PROGRAM LsBkgrdLsSerialCom
VAR_INPUT
	Config : LightspeedConfig;
END_VAR
VAR
END_VAR

// AttenuationFilterConfigs
IF Config.AttenuationFilterConfigs.FW212CAttenuationFilterConfig.IsEnabled OR 
   Config.AttenuationFilterConfigs.ELL14kAttenuationFilterConfig.IsEnabled OR
   Config.AttenuationFilterConfigs.ELL9AttenuationFilterConfig.IsEnabled THEN
	BkgrdSerialAttenuation();	
END_IF

// SliderAttenuationFilterConfigs
IF Config.SliderAttenuationFilterConfigs.ELL6SliderFilterConfig.IsEnabled THEN
	BkgrdSerialSliderAttenuation();	
END_IF

// RotatingSwitchConfigs
IF Config.RotatingSwitchConfigs.ELL18RotatingSwitchConfig.IsEnabled THEN
	BkgrdSerialRotatingSwitch();	
END_IF

// PolarisationFilterConfigs
IF Config.PolarisationFilterConfigs.FW212CPolarisationFilterConfig.IsEnabled OR 
   Config.PolarisationFilterConfigs.ELL14KPolarisationFilterConfig.IsEnabled THEN
	BkgrdSerialPolarisation();		
END_IF

// LaserConfigs
IF Config.LaserConfigs.SMD12LaserConfig.IsEnabled OR 
	Config.LaserConfigs.Sapphire488LaserConfig.IsEnabled THEN
	BkgrdSerialLaser();
END_IF

// FiberSwitchConfigs
IF Config.FiberSwitchConfigs.EOLFiberSwitchConfig.IsEnabled THEN
	BkgrdSerialFiberSwitch();
END_IF

// OpticalPowermeterConfigs
IF Config.OpticalPowermeterConfigs.PM101OpticalPowermeterConfigHs.IsEnabled THEN
	BkgrdSerialOpticalPowermeterHs();	
END_IF
IF Config.OpticalPowermeterConfigs.PM101OpticalPowermeterConfigHt.IsEnabled THEN
	BkgrdSerialOpticalPowermeterHt();	
END_IF

// MppcConfigs
IF Config.MppcConfigs.C13336MppcConfigWide.IsEnabled THEN
	BkgrdSerialMppcWide();
END_IF
IF Config.MppcConfigs.C13336MppcConfigNarrow.IsEnabled THEN
	BkgrdSerialMppcNarrow();
END_IF

END_PROGRAM

(* stored: Version 1.1.0.1, ProductVersion 3.1.4024.12
   POU LsBkgrdLsSerialCom: Id {6c01a632-fa48-42a1-9afe-d9e39229f4f6}, SpecialFunc None *)
